(*
SPDX-FileCopyrightText: © 2026 Oleksandr Tiutyk <trofimich@gmail.com>
SPDX-License-Identifier: MIT
License: https://opensource.org/license/mit
*)

{attribute 'no_explicit_call' := 'do not call this function block directly'} 
PROGRAM SignedInt64
VAR CONSTANT
	MIN_VALUE : LINT := -9_223_372_036_854_775_808;
	MAX_VALUE : LINT := +9_223_372_036_854_775_807;
END_VAR
VAR
	{attribute 'hide'} 
	_ClassName : STRING := __POUNAME();
END_VAR

{attribute 'monitoring' := 'call'}
PROPERTY ClassName : REFERENCE TO STRING
GET
ClassName REF= _ClassName;
END_GET
END_PROPERTY

{attribute 'monitoring' := 'call'}
PROPERTY NamespaceName : REFERENCE TO STRING
GET
NamespaceName REF= CurrentNamespace.Name;
END_GET
END_PROPERTY

END_PROGRAM

(* stored: Version 1.1.0.1
   POU SignedInt64: Id {fda2daf2-422d-481e-b127-7b1b7aaf3ced}, SpecialFunc None
   Property ClassName: Id {73c2a366-2fd1-492d-893d-96b5466242bd}
   Get Get: Id {631facea-e6d0-4316-8c24-d4e56dfca243}
   Property NamespaceName: Id {cd33d955-51ac-4fa8-b782-ec1764ca8c2b}
   Get Get: Id {ab637efb-6fa0-4b4e-87f8-3bdaddbe4e54} *)
